// TIA Portal V20 export
TYPE "typeIntConditionHmiInterface"
// stored: Access Published, Namespace Unit1.Em13
   STRUCT
      Axis_18 { S7_SetPoint := 'True'} : "LER_typeAxisIntlockAll";   // JrUnloadingX
      Axis_19 { S7_SetPoint := 'True'} : "LER_typeAxisIntlockAll";   // JrUnloadingZ
      Axis_20 { S7_SetPoint := 'True'} : "LER_typeAxisIntlockAll";   // JrUnloadingC
      Actuator_68 { S7_SetPoint := 'True'} : "LER_typeAxisActuatorCondition";   // AnodeNgBoxLockUpDown
   END_STRUCT;
END_TYPE
